TYPE ST_HIERARCHYDATACS :
STRUCT
	UNITQTY		:STRING;
	GTIN		:STRING;
	EAN			:STRING;
END_STRUCT
END_TYPE

(* stored: Version 1.1.0.1, ProductVersion 3.1.4024.13
   DUT ST_HIERARCHYDATACS: Id {aaadd1c1-9402-46dc-9be0-ee752b2de4c5} *)
